// TIA Portal project "ReconocimientoObjetos" (V18)
// Vorlageprojekt für das Buch mit Zielsystem S7-1200

(* hardware
DEVICE "S7-1200-Station_1"  S7-1200 Station
   slot 0: "Baugruppenträger_0"  Rack  V1.0
   slot 1: "PLC_1"  CPU 1211C DC/DC/DC  6ES7 211-1AE40-0XB0  V4.1
*)

// ===== PLC "PLC_1"  CPU 1211C DC/DC/DC =====

VAR_GLOBAL   // PLC tag table "Standard-Variablentabelle"
   "sensorInductivo" AT %I0.0 : Bool;   // Sensor que reconoce los objetos de metal
   "sensorCapacitivo" AT %I0.1 : Bool;   // Sensor que reconoce los objetos de plastico
   "sensorCilindro" AT %I0.2 : Bool;   // Sensor del Cilindro
   "infrarrojoFinalPlastico" AT %I0.3 : Bool;   // Sensor final de la cinta de objetos de plastico
   "infrarrojoFinalMetal" AT %I0.4 : Bool;   // Sensor final de la cinta de objetos de metal
   "cintaPrincipal" AT %Q0.0 : Bool;   // Motor de la cinta transportadora principal
   "cintaPlastico" AT %Q0.1 : Bool;   // Motor de la cinta transportadora de objetos de plastico
   "cintaMetal" AT %Q0.2 : Bool;   // Motor de la cinta transportadora de objetos de metal
   "cilindro" AT %Q0.3 : Bool;   // Activacion del cilindro
   "marcaCintaPrincipal" AT %M80.0 : Bool;
   "marcaMoverObjeto" AT %M80.1 : Bool;
   "marcaCintaPlastico" AT %M80.2 : Bool;
   "marcaCintaMetal" AT %M80.3 : Bool;
   "marcaObjetoPlastico" AT %M80.4 : Bool;
   "marcaObjetoMetal" AT %M80.5 : Bool;
   "marcaFN1" AT %M90.0 : Bool;
   "marcaFN2" AT %M90.1 : Bool;
   "marcaFN3" AT %M90.2 : Bool;
   "marcaFN4" AT %M90.3 : Bool;
   "marcaFN5" AT %M90.4 : Bool;
END_VAR

ORGANIZATION_BLOCK "Main"   // OB1, LAD, ProgramCycle
TITLE = "Main Program Sweep (Cycle)"
{ S7_Optimized_Access := 'TRUE' }
VERSION : 0.1
   VAR_INPUT
      Initial_Call : Bool;   // Initial call of this OB
      Remanence : Bool;   // =True, if remanent data are available
   END_VAR
   VAR_TEMP   // added for the SCL form of the ladder/FBD networks
      _w1 : Bool;
   END_VAR
BEGIN

REGION Network 1: Ihr Programm / Primer objeto por la cinta transportadora
   // Schreiben Sie ab Netzwerk 2 Ihr Programm
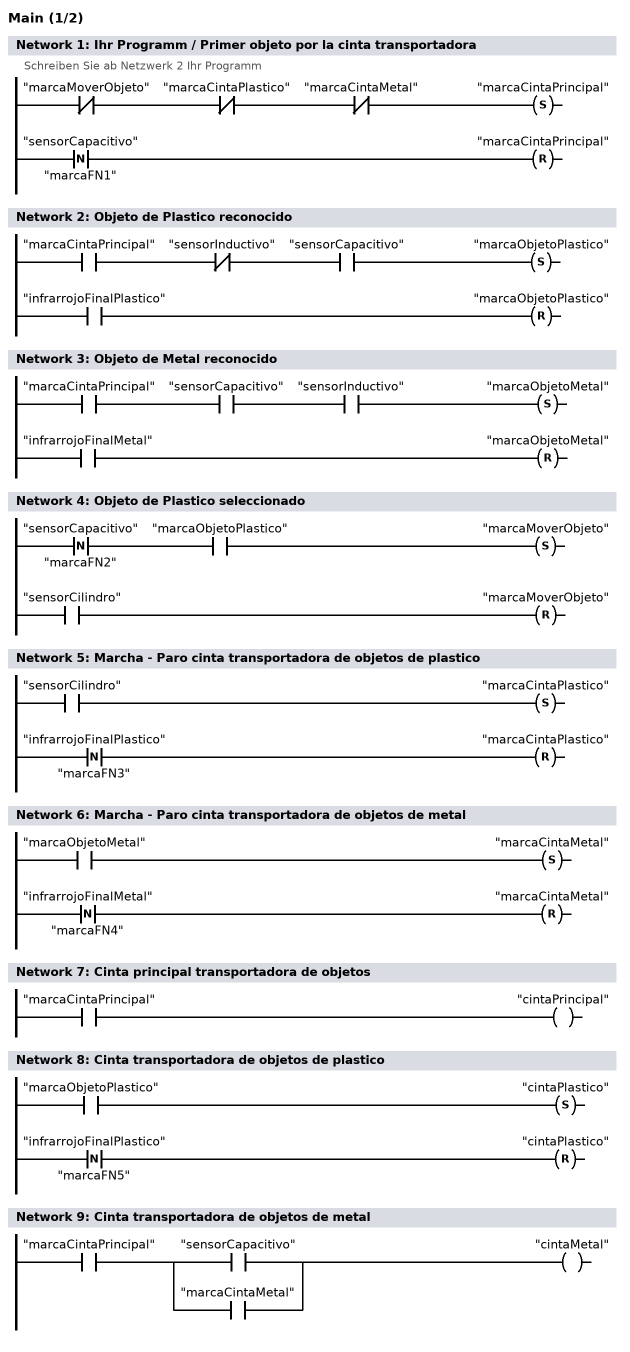
   RUNG wire#powerrail
      I_Contact( "marcaMoverObjeto" )
      I_Contact( "marcaCintaPlastico" )
      I_Contact( "marcaCintaMetal" )
      S_Coil( "marcaCintaPrincipal" )
   END_RUNG
   RUNG wire#powerrail
      N_Contact(operand := "sensorCapacitivo", bit := "marcaFN1")
      R_Coil( "marcaCintaPrincipal" )
   END_RUNG
   // the same network as SCL:
   IF NOT "marcaMoverObjeto" AND NOT "marcaCintaPlastico" AND NOT "marcaCintaMetal" THEN
       "marcaCintaPrincipal" := TRUE;
   END_IF;
   #_w1 := NOT "sensorCapacitivo" AND "marcaFN1";   // falling edge of "sensorCapacitivo"
   "marcaFN1" := "sensorCapacitivo";
   IF #_w1 THEN "marcaCintaPrincipal" := FALSE; END_IF;
END_REGION

REGION Network 2: Objeto de Plastico reconocido
   RUNG wire#powerrail
      Contact( "marcaCintaPrincipal" )
      I_Contact( "sensorInductivo" )
      Contact( "sensorCapacitivo" )
      S_Coil( "marcaObjetoPlastico" )
   END_RUNG
   RUNG wire#powerrail
      Contact( "infrarrojoFinalPlastico" )
      R_Coil( "marcaObjetoPlastico" )
   END_RUNG
   // the same network as SCL:
   IF "marcaCintaPrincipal" AND NOT "sensorInductivo" AND "sensorCapacitivo" THEN
       "marcaObjetoPlastico" := TRUE;
   END_IF;
   IF "infrarrojoFinalPlastico" THEN "marcaObjetoPlastico" := FALSE; END_IF;
END_REGION

REGION Network 3: Objeto de Metal reconocido
   RUNG wire#powerrail
      Contact( "marcaCintaPrincipal" )
      Contact( "sensorCapacitivo" )
      Contact( "sensorInductivo" )
      S_Coil( "marcaObjetoMetal" )
   END_RUNG
   RUNG wire#powerrail
      Contact( "infrarrojoFinalMetal" )
      R_Coil( "marcaObjetoMetal" )
   END_RUNG
   // the same network as SCL:
   IF "marcaCintaPrincipal" AND "sensorCapacitivo" AND "sensorInductivo" THEN
       "marcaObjetoMetal" := TRUE;
   END_IF;
   IF "infrarrojoFinalMetal" THEN "marcaObjetoMetal" := FALSE; END_IF;
END_REGION

REGION Network 4: Objeto de Plastico seleccionado
   RUNG wire#powerrail
      N_Contact(operand := "sensorCapacitivo", bit := "marcaFN2")
      Contact( "marcaObjetoPlastico" )
      S_Coil( "marcaMoverObjeto" )
   END_RUNG
   RUNG wire#powerrail
      Contact( "sensorCilindro" )
      R_Coil( "marcaMoverObjeto" )
   END_RUNG
   // the same network as SCL:
   #_w1 := NOT "sensorCapacitivo" AND "marcaFN2";   // falling edge of "sensorCapacitivo"
   "marcaFN2" := "sensorCapacitivo";
   IF #_w1 AND "marcaObjetoPlastico" THEN "marcaMoverObjeto" := TRUE; END_IF;
   IF "sensorCilindro" THEN "marcaMoverObjeto" := FALSE; END_IF;
END_REGION

REGION Network 5: Marcha - Paro cinta transportadora de objetos de plastico
   RUNG wire#powerrail
      Contact( "sensorCilindro" )
      S_Coil( "marcaCintaPlastico" )
   END_RUNG
   RUNG wire#powerrail
      N_Contact(operand := "infrarrojoFinalPlastico", bit := "marcaFN3")
      R_Coil( "marcaCintaPlastico" )
   END_RUNG
   // the same network as SCL:
   IF "sensorCilindro" THEN "marcaCintaPlastico" := TRUE; END_IF;
   #_w1 := NOT "infrarrojoFinalPlastico" AND "marcaFN3";   // falling edge of "infrarrojoFinalPlastico"
   "marcaFN3" := "infrarrojoFinalPlastico";
   IF #_w1 THEN "marcaCintaPlastico" := FALSE; END_IF;
END_REGION

REGION Network 6: Marcha - Paro cinta transportadora de objetos de metal
   RUNG wire#powerrail
      Contact( "marcaObjetoMetal" )
      S_Coil( "marcaCintaMetal" )
   END_RUNG
   RUNG wire#powerrail
      N_Contact(operand := "infrarrojoFinalMetal", bit := "marcaFN4")
      R_Coil( "marcaCintaMetal" )
   END_RUNG
   // the same network as SCL:
   IF "marcaObjetoMetal" THEN "marcaCintaMetal" := TRUE; END_IF;
   #_w1 := NOT "infrarrojoFinalMetal" AND "marcaFN4";   // falling edge of "infrarrojoFinalMetal"
   "marcaFN4" := "infrarrojoFinalMetal";
   IF #_w1 THEN "marcaCintaMetal" := FALSE; END_IF;
END_REGION

REGION Network 7: Cinta principal transportadora de objetos
   RUNG wire#powerrail
      Contact( "marcaCintaPrincipal" )
      Coil( "cintaPrincipal" )
   END_RUNG
   // the same network as SCL:
   "cintaPrincipal" := "marcaCintaPrincipal";
END_REGION

REGION Network 8: Cinta transportadora de objetos de plastico
   RUNG wire#powerrail
      Contact( "marcaObjetoPlastico" )
      S_Coil( "cintaPlastico" )
   END_RUNG
   RUNG wire#powerrail
      N_Contact(operand := "infrarrojoFinalPlastico", bit := "marcaFN5")
      R_Coil( "cintaPlastico" )
   END_RUNG
   // the same network as SCL:
   IF "marcaObjetoPlastico" THEN "cintaPlastico" := TRUE; END_IF;
   #_w1 := NOT "infrarrojoFinalPlastico" AND "marcaFN5";   // falling edge of "infrarrojoFinalPlastico"
   "marcaFN5" := "infrarrojoFinalPlastico";
   IF #_w1 THEN "cintaPlastico" := FALSE; END_IF;
END_REGION

REGION Network 9: Cinta transportadora de objetos de metal
   RUNG wire#powerrail
      Contact( "marcaCintaPrincipal" )
      wire#w1
      Contact( "sensorCapacitivo" )
      wire#w2
      Coil( "cintaMetal" )
   END_RUNG
   RUNG wire#w1
      Contact( "marcaCintaMetal" )
   END_RUNG wire#w2
   // the same network as SCL:
   "cintaMetal" := "marcaCintaPrincipal" AND ("sensorCapacitivo" OR "marcaCintaMetal");
END_REGION

REGION Network 10: Cilindro Activo
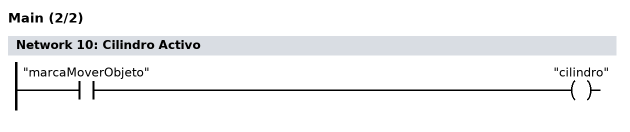
   RUNG wire#powerrail
      Contact( "marcaMoverObjeto" )
      Coil( "cilindro" )
   END_RUNG
   // the same network as SCL:
   "cilindro" := "marcaMoverObjeto";
END_REGION
END_ORGANIZATION_BLOCK